# EPICS SNL sequencer program: acq400iocApp/src/aoRangeSet.stt
/*************************************************************************\
ao420_range_set.st : rescale AO records depending on range.
\*************************************************************************/
program ao420_range_set
option +r;

int ref;	assign ref to "{UUT}:{SITE}:AO:REF";
int gain;	assign gain to "{UUT}:{SITE}:AO:GAIN:CH:{CID}";

double drvl;	assign drvl to "{UUT}:{SITE}:AO:SLOW_SET:CH:{CID}.DRVL";
double drvh;	assign drvh to "{UUT}:{SITE}:AO:SLOW_SET:CH:{CID}.DRVH";
double eslo;	assign eslo to "{UUT}:{SITE}:AO:SLOW_SET:CH:{CID}.ESLO";
double hopr;	assign hopr to "{UUT}:{SITE}:AO:SLOW_SET:CH:{CID}.HOPR";
double lopr;	assign lopr to "{UUT}:{SITE}:AO:SLOW_SET:CH:{CID}.LOPR";
double val;	assign val  to "{UUT}:{SITE}:AO:SLOW_SET:CH:{CID}";
int data32;     assign data32 to "{UUT}:{SITE}:data32";

string model;	assign model to "{UUT}:{SITE}:MODEL";

monitor ref;
monitor gain;

int ref0;
int gain0;

double denom = 65535;

int first_time = 1;

ss gain_set
{
	state init {
		when() {
			ref0 = ref;
			gain0 = gain;
			pvGet(model);
			pvGet(data32);
			if (data32){
				denom = 0xffffffffU;
			}

			/* AO420FMC and AO422 is always fixed 5V */
			if (strncmp(model, "AO420FMC", 8) == 0 ||
			    strncmp(model, "AO422",    5) == 0){
				ref0 = ref = 1;
				pvPut(ref);
			}
		} state run
	}
	state run
	{
		when(first_time || ref != ref0 || gain != gain0){
			if (ref==0 && gain==0){
				drvl = lopr = -2.5;
				drvh = hopr = 2.4999;
			}else if (ref==1 && gain==1){
				drvl = lopr = -10;
				drvh = hopr = 9.9999;
			}else{
				drvl = lopr = -5;
				drvh = hopr = 4.9999;
			}
			eslo = (hopr - lopr) / denom;
			printf("%s lo %.2f hi %.2f eslo %.2e\n", macValueGet("CID"), drvl, drvh, eslo);
			pvPut(drvl);
			pvPut(drvh);
			pvPut(eslo);
			pvPut(hopr);
			pvPut(lopr);
			val = 0;
			pvPut(val);
			first_time = 0;
			ref0 = ref;
			gain0 = gain;
		} state run
	}
}
